SUBAPPLICATION Uebung_004 (* Subapplication Type *)
  (* Standard: 61499-2 *)
  (* Version 1.0, 2023-10-23, franz *)
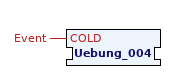
  EVENT_INPUT
    COLD;
  END_EVENT
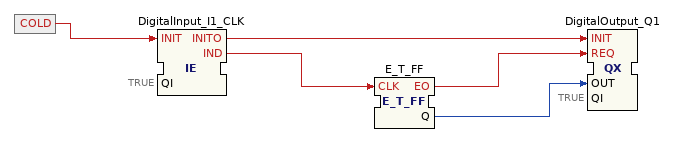
  FBS
    DigitalOutput_Q1 : QX(QI := TRUE);
    DigitalInput_I1_CLK : IE(QI := TRUE);
    E_T_FF : E_T_FF;
  END_FBS
  EVENT_CONNECTIONS
    COLD TO DigitalInput_I1_CLK.INIT;
    DigitalInput_I1_CLK.INITO TO DigitalOutput_Q1.INIT;
    DigitalInput_I1_CLK.IND TO E_T_FF.CLK;
    E_T_FF.EO TO DigitalOutput_Q1.REQ;
  END_CONNECTIONS
  DATA_CONNECTIONS
    E_T_FF.Q TO DigitalOutput_Q1.OUT;
  END_CONNECTIONS
END_SUBAPPLICATION
